FUNCTION_BLOCK Top
  (* Standard: 61499-2 *)
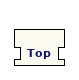
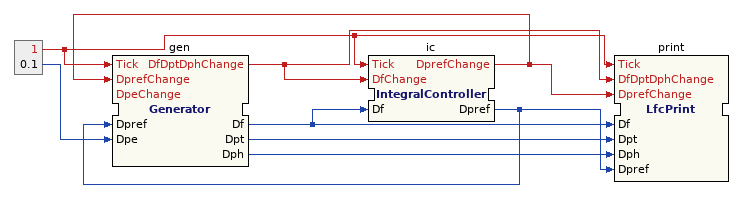
  FBS
    gen : Generator;
    ic : IntegralController;
    print : LfcPrint;
  END_FBS
  EVENT_CONNECTIONS
    1 TO ic.Tick;
    1 TO gen.Tick;
    1 TO print.Tick;
    gen.DfDptDphChange TO ic.DfChange;
    ic.DprefChange TO gen.DprefChange;
    gen.DfDptDphChange TO print.DfDptDphChange;
    ic.DprefChange TO print.DprefChange;
  END_CONNECTIONS
  DATA_CONNECTIONS
    gen.Df TO ic.Df;
    ic.Dpref TO gen.Dpref;
    0.1 TO gen.Dpe;
    gen.Df TO print.Df;
    gen.Dpt TO print.Dpt;
    gen.Dph TO print.Dph;
    ic.Dpref TO print.Dpref;
  END_CONNECTIONS
END_FUNCTION_BLOCK
